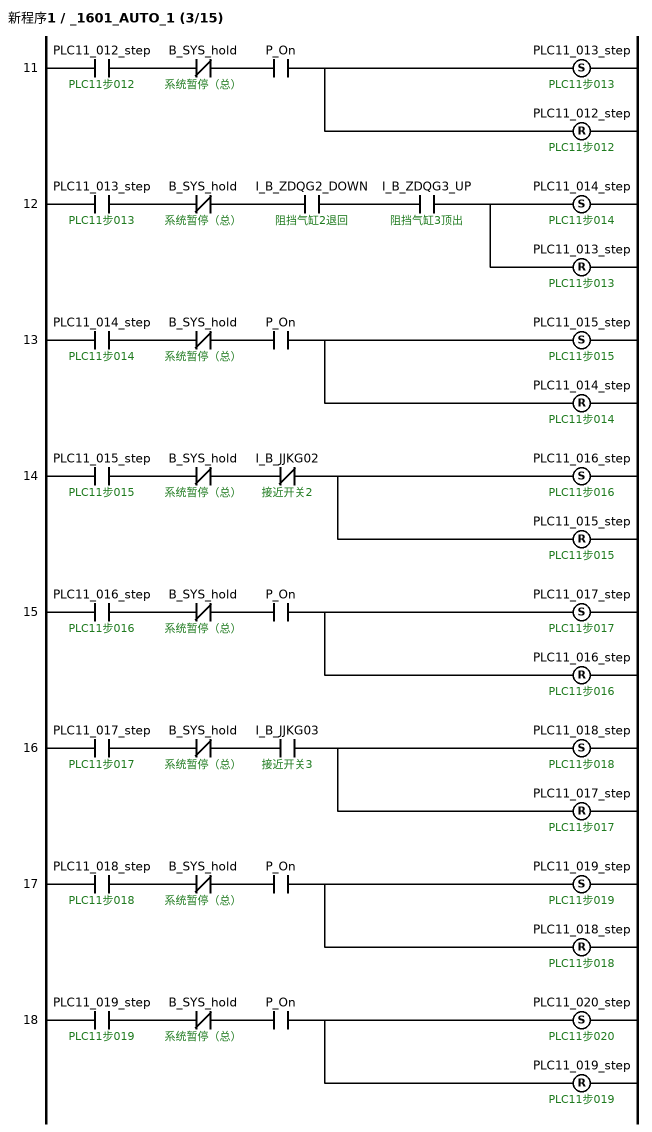
; [picture p24: 新程序1 / _1601_AUTO_1, rungs 11-18]
; rung 11
LD PLC11_012_step  ; PLC11步012
ANDNOT B_SYS_hold  ; 系统暂停（总）
AND P_On
SET PLC11_013_step  ; PLC11步013
RSET PLC11_012_step  ; PLC11步012
; rung 12
LD PLC11_013_step  ; PLC11步013
ANDNOT B_SYS_hold  ; 系统暂停（总）
AND I_B_ZDQG2_DOWN  ; 阻挡气缸2退回
AND I_B_ZDQG3_UP  ; 阻挡气缸3顶出
SET PLC11_014_step  ; PLC11步014
RSET PLC11_013_step  ; PLC11步013
; rung 13
LD PLC11_014_step  ; PLC11步014
ANDNOT B_SYS_hold  ; 系统暂停（总）
AND P_On
SET PLC11_015_step  ; PLC11步015
RSET PLC11_014_step  ; PLC11步014
; rung 14
LD PLC11_015_step  ; PLC11步015
ANDNOT B_SYS_hold  ; 系统暂停（总）
ANDNOT I_B_JJKG02  ; 接近开关2
SET PLC11_016_step  ; PLC11步016
RSET PLC11_015_step  ; PLC11步015
; rung 15
LD PLC11_016_step  ; PLC11步016
ANDNOT B_SYS_hold  ; 系统暂停（总）
AND P_On
SET PLC11_017_step  ; PLC11步017
RSET PLC11_016_step  ; PLC11步016
; rung 16
LD PLC11_017_step  ; PLC11步017
ANDNOT B_SYS_hold  ; 系统暂停（总）
AND I_B_JJKG03  ; 接近开关3
SET PLC11_018_step  ; PLC11步018
RSET PLC11_017_step  ; PLC11步017
; rung 17
LD PLC11_018_step  ; PLC11步018
ANDNOT B_SYS_hold  ; 系统暂停（总）
AND P_On
SET PLC11_019_step  ; PLC11步019
RSET PLC11_018_step  ; PLC11步018
; rung 18
LD PLC11_019_step  ; PLC11步019
ANDNOT B_SYS_hold  ; 系统暂停（总）
AND P_On
SET PLC11_020_step  ; PLC11步020
RSET PLC11_019_step  ; PLC11步019

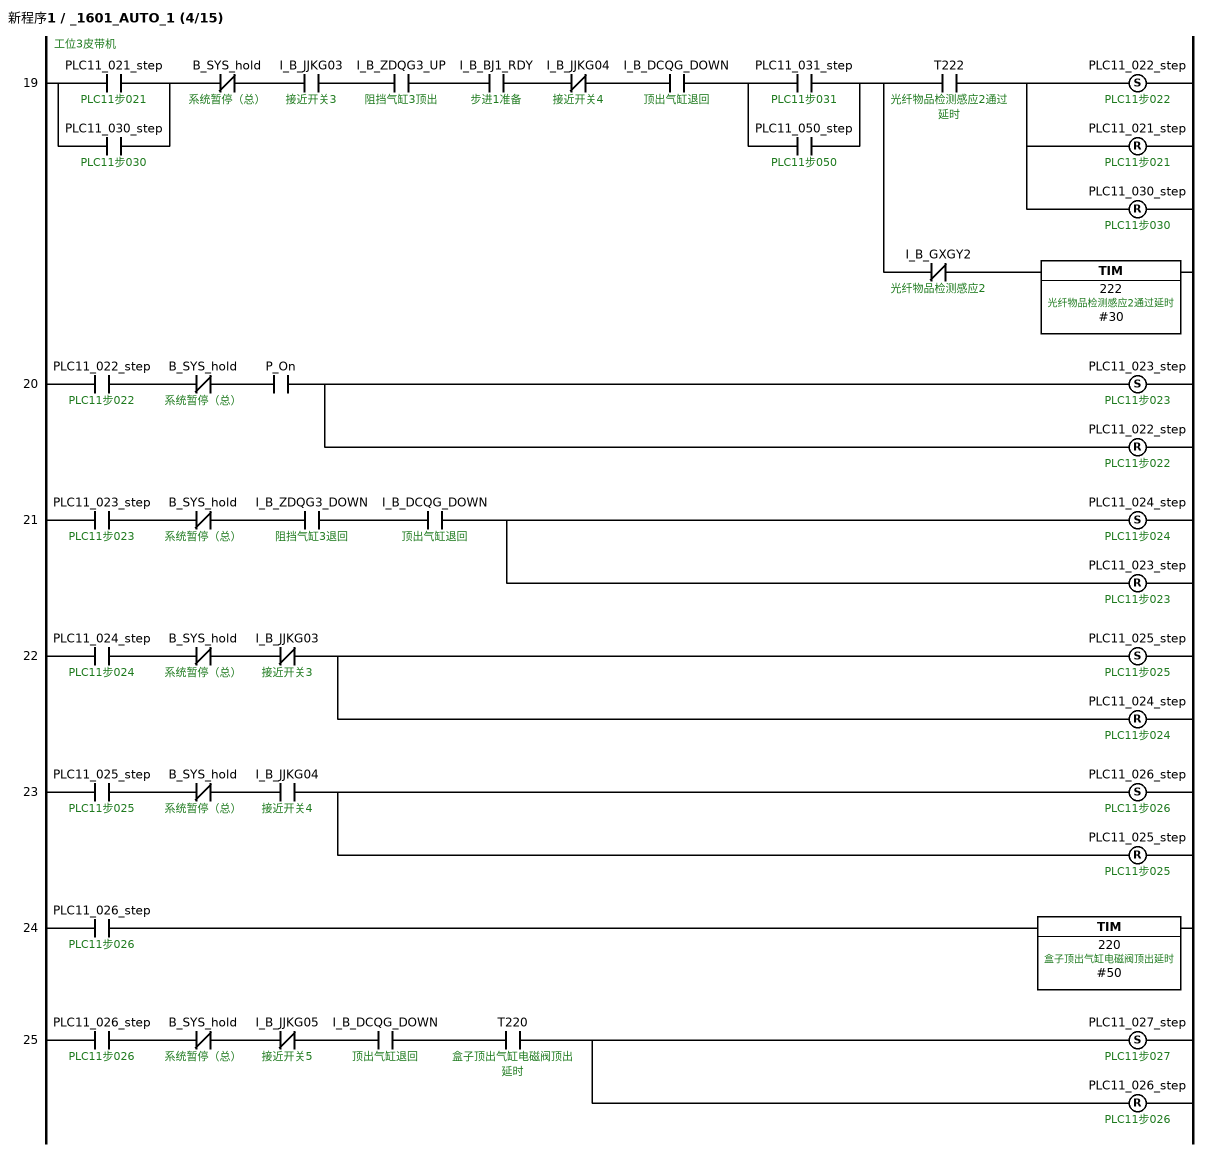
; rung 19: 工位3皮带机
LD PLC11_021_step  ; PLC11步021
OR PLC11_030_step  ; PLC11步030
ANDNOT B_SYS_hold  ; 系统暂停（总）
AND I_B_JJKG03  ; 接近开关3
AND I_B_ZDQG3_UP  ; 阻挡气缸3顶出
AND I_B_BJ1_RDY  ; 步进1准备
ANDNOT I_B_JJKG04  ; 接近开关4
AND I_B_DCQG_DOWN  ; 顶出气缸退回
LD PLC11_031_step  ; PLC11步031
OR PLC11_050_step  ; PLC11步050
ANDLD
OUT TR0
AND T222  ; 光纤物品检测感应2通过延时
SET PLC11_022_step  ; PLC11步022
RSET PLC11_021_step  ; PLC11步021
RSET PLC11_030_step  ; PLC11步030
LD TR0
ANDNOT I_B_GXGY2  ; 光纤物品检测感应2
TIM 222 #30  ; 光纤物品检测感应2通过延时
; rung 20
LD PLC11_022_step  ; PLC11步022
ANDNOT B_SYS_hold  ; 系统暂停（总）
AND P_On
SET PLC11_023_step  ; PLC11步023
RSET PLC11_022_step  ; PLC11步022
; rung 21
LD PLC11_023_step  ; PLC11步023
ANDNOT B_SYS_hold  ; 系统暂停（总）
AND I_B_ZDQG3_DOWN  ; 阻挡气缸3退回
AND I_B_DCQG_DOWN  ; 顶出气缸退回
SET PLC11_024_step  ; PLC11步024
RSET PLC11_023_step  ; PLC11步023
; rung 22
LD PLC11_024_step  ; PLC11步024
ANDNOT B_SYS_hold  ; 系统暂停（总）
ANDNOT I_B_JJKG03  ; 接近开关3
SET PLC11_025_step  ; PLC11步025
RSET PLC11_024_step  ; PLC11步024
; rung 23
LD PLC11_025_step  ; PLC11步025
ANDNOT B_SYS_hold  ; 系统暂停（总）
AND I_B_JJKG04  ; 接近开关4
SET PLC11_026_step  ; PLC11步026
RSET PLC11_025_step  ; PLC11步025
; rung 24
LD PLC11_026_step  ; PLC11步026
TIM 220 #50  ; 盒子顶出气缸电磁阀顶出延时
; rung 25
LD PLC11_026_step  ; PLC11步026
ANDNOT B_SYS_hold  ; 系统暂停（总）
ANDNOT I_B_JJKG05  ; 接近开关5
AND I_B_DCQG_DOWN  ; 顶出气缸退回
AND T220  ; 盒子顶出气缸电磁阀顶出延时
SET PLC11_027_step  ; PLC11步027
RSET PLC11_026_step  ; PLC11步026

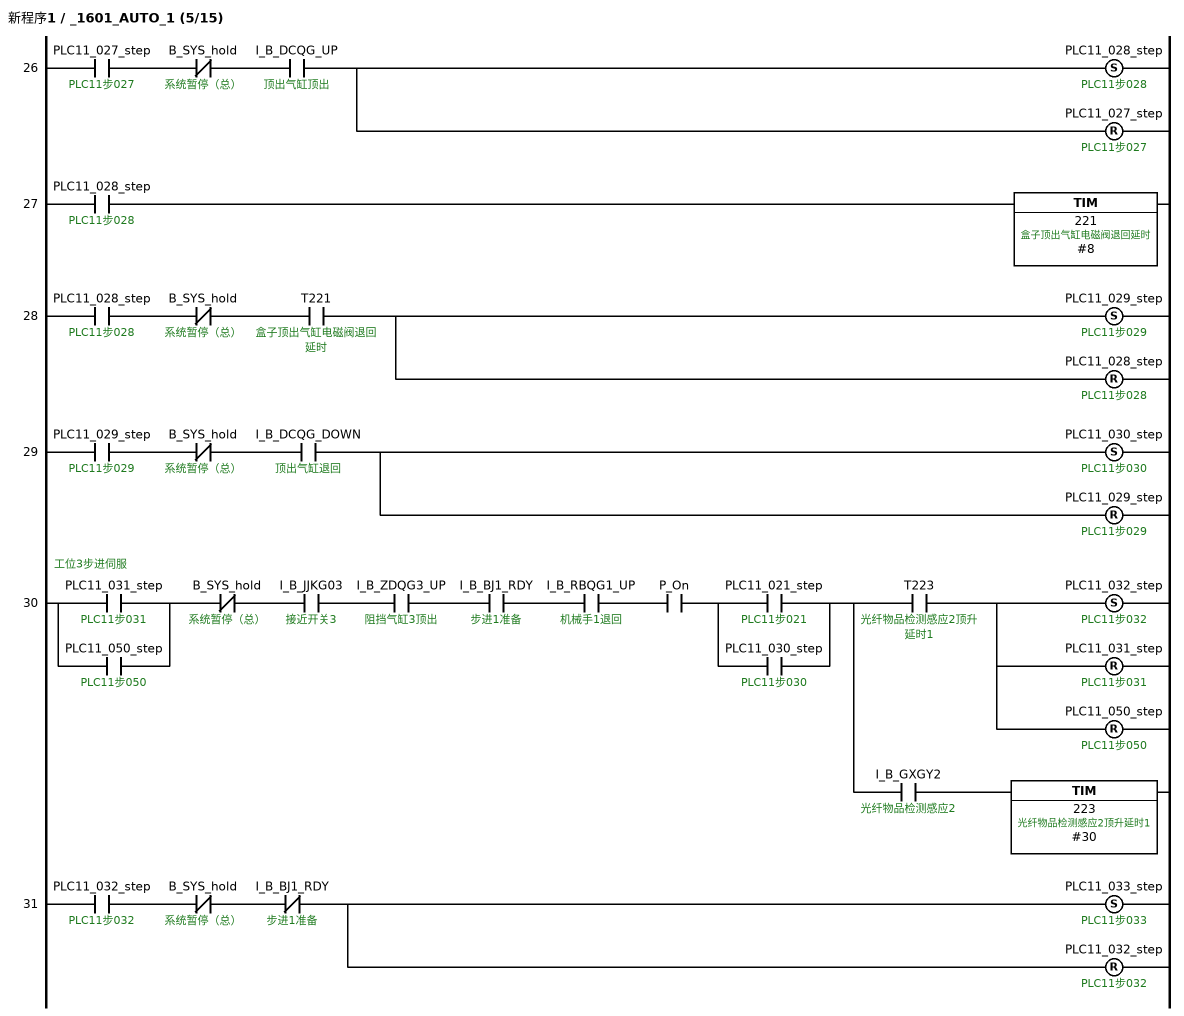
; rung 26
LD PLC11_027_step  ; PLC11步027
ANDNOT B_SYS_hold  ; 系统暂停（总）
AND I_B_DCQG_UP  ; 顶出气缸顶出
SET PLC11_028_step  ; PLC11步028
RSET PLC11_027_step  ; PLC11步027
; rung 27
LD PLC11_028_step  ; PLC11步028
TIM 221 #8  ; 盒子顶出气缸电磁阀退回延时
; rung 28
LD PLC11_028_step  ; PLC11步028
ANDNOT B_SYS_hold  ; 系统暂停（总）
AND T221  ; 盒子顶出气缸电磁阀退回延时
SET PLC11_029_step  ; PLC11步029
RSET PLC11_028_step  ; PLC11步028
; rung 29
LD PLC11_029_step  ; PLC11步029
ANDNOT B_SYS_hold  ; 系统暂停（总）
AND I_B_DCQG_DOWN  ; 顶出气缸退回
SET PLC11_030_step  ; PLC11步030
RSET PLC11_029_step  ; PLC11步029
; rung 30: 工位3步进伺服
LD PLC11_031_step  ; PLC11步031
OR PLC11_050_step  ; PLC11步050
ANDNOT B_SYS_hold  ; 系统暂停（总）
AND I_B_JJKG03  ; 接近开关3
AND I_B_ZDQG3_UP  ; 阻挡气缸3顶出
AND I_B_BJ1_RDY  ; 步进1准备
AND I_B_RBQG1_UP  ; 机械手1退回
AND P_On
LD PLC11_021_step  ; PLC11步021
OR PLC11_030_step  ; PLC11步030
ANDLD
OUT TR0
AND T223  ; 光纤物品检测感应2顶升延时1
SET PLC11_032_step  ; PLC11步032
RSET PLC11_031_step  ; PLC11步031
RSET PLC11_050_step  ; PLC11步050
LD TR0
AND I_B_GXGY2  ; 光纤物品检测感应2
TIM 223 #30  ; 光纤物品检测感应2顶升延时1
; rung 31
LD PLC11_032_step  ; PLC11步032
ANDNOT B_SYS_hold  ; 系统暂停（总）
ANDNOT I_B_BJ1_RDY  ; 步进1准备
SET PLC11_033_step  ; PLC11步033
RSET PLC11_032_step  ; PLC11步032

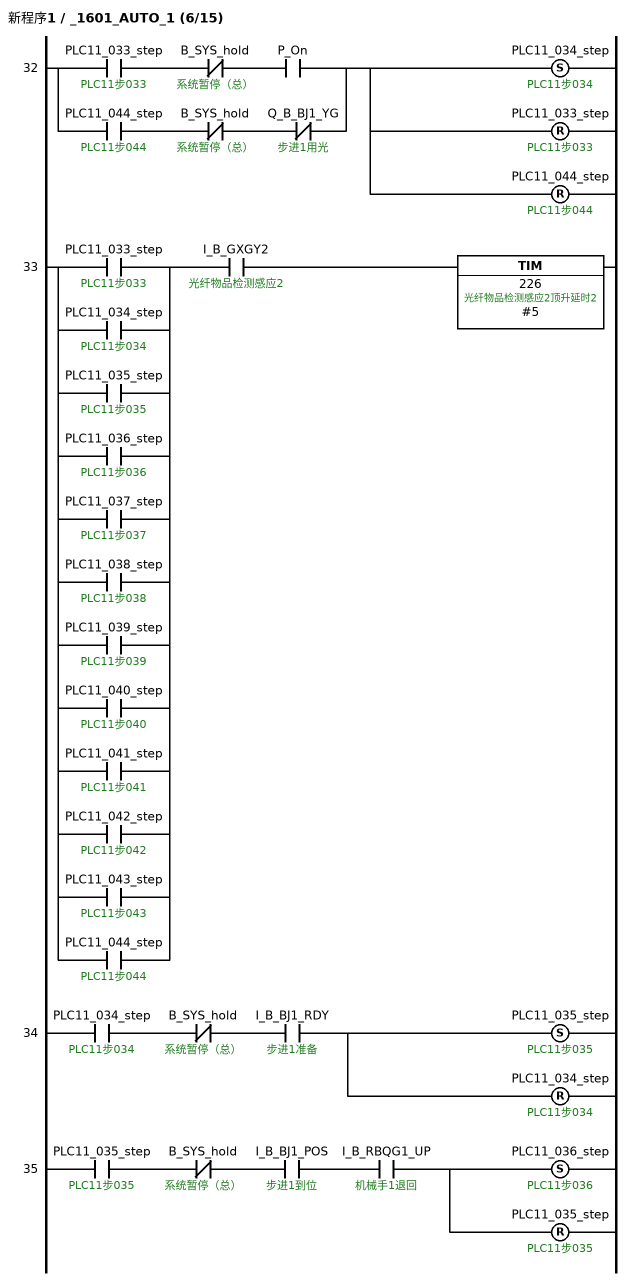
; rung 32
LD PLC11_033_step  ; PLC11步033
ANDNOT B_SYS_hold  ; 系统暂停（总）
AND P_On
LD PLC11_044_step  ; PLC11步044
ANDNOT B_SYS_hold  ; 系统暂停（总）
ANDNOT Q_B_BJ1_YG  ; 步进1用光
ORLD
SET PLC11_034_step  ; PLC11步034
RSET PLC11_033_step  ; PLC11步033
RSET PLC11_044_step  ; PLC11步044
; rung 33
LD PLC11_033_step  ; PLC11步033
OR PLC11_034_step  ; PLC11步034
OR PLC11_035_step  ; PLC11步035
OR PLC11_036_step  ; PLC11步036
OR PLC11_037_step  ; PLC11步037
OR PLC11_038_step  ; PLC11步038
OR PLC11_039_step  ; PLC11步039
OR PLC11_040_step  ; PLC11步040
OR PLC11_041_step  ; PLC11步041
OR PLC11_042_step  ; PLC11步042
OR PLC11_043_step  ; PLC11步043
OR PLC11_044_step  ; PLC11步044
AND I_B_GXGY2  ; 光纤物品检测感应2
TIM 226 #5  ; 光纤物品检测感应2顶升延时2
; rung 34
LD PLC11_034_step  ; PLC11步034
ANDNOT B_SYS_hold  ; 系统暂停（总）
AND I_B_BJ1_RDY  ; 步进1准备
SET PLC11_035_step  ; PLC11步035
RSET PLC11_034_step  ; PLC11步034
; rung 35
LD PLC11_035_step  ; PLC11步035
ANDNOT B_SYS_hold  ; 系统暂停（总）
AND I_B_BJ1_POS  ; 步进1到位
AND I_B_RBQG1_UP  ; 机械手1退回
SET PLC11_036_step  ; PLC11步036
RSET PLC11_035_step  ; PLC11步035

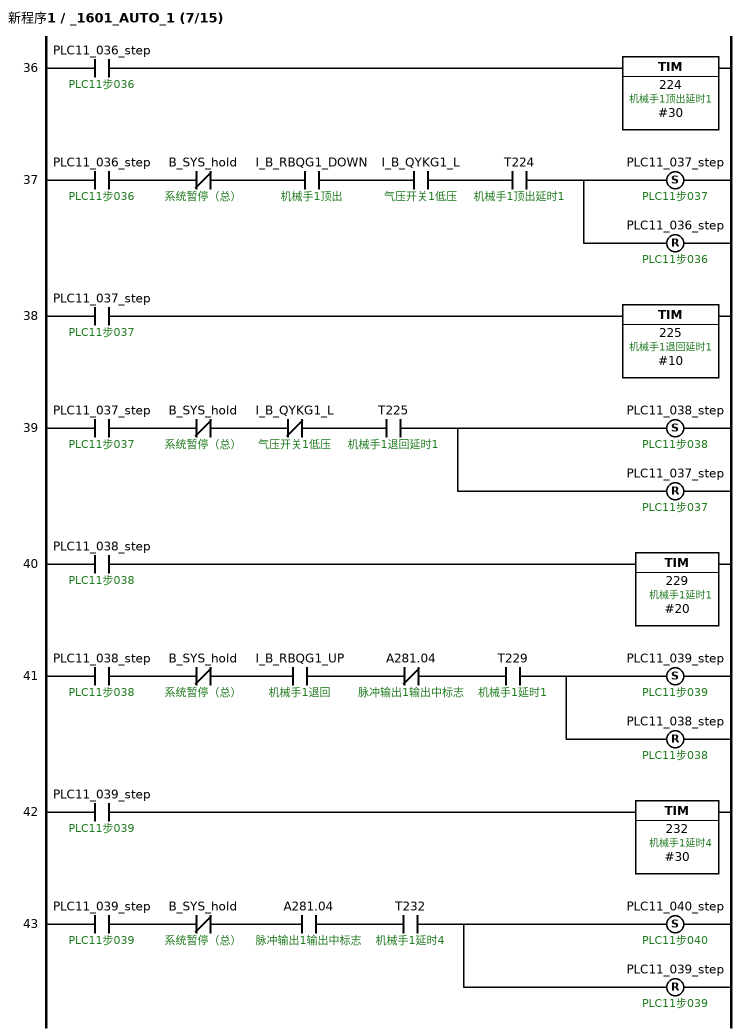
; rung 36
LD PLC11_036_step  ; PLC11步036
TIM 224 #30  ; 机械手1顶出延时1
; rung 37
LD PLC11_036_step  ; PLC11步036
ANDNOT B_SYS_hold  ; 系统暂停（总）
AND I_B_RBQG1_DOWN  ; 机械手1顶出
AND I_B_QYKG1_L  ; 气压开关1低压
AND T224  ; 机械手1顶出延时1
SET PLC11_037_step  ; PLC11步037
RSET PLC11_036_step  ; PLC11步036
; rung 38
LD PLC11_037_step  ; PLC11步037
TIM 225 #10  ; 机械手1退回延时1
; rung 39
LD PLC11_037_step  ; PLC11步037
ANDNOT B_SYS_hold  ; 系统暂停（总）
ANDNOT I_B_QYKG1_L  ; 气压开关1低压
AND T225  ; 机械手1退回延时1
SET PLC11_038_step  ; PLC11步038
RSET PLC11_037_step  ; PLC11步037
; rung 40
LD PLC11_038_step  ; PLC11步038
TIM 229 #20  ; 机械手1延时1
; rung 41
LD PLC11_038_step  ; PLC11步038
ANDNOT B_SYS_hold  ; 系统暂停（总）
AND I_B_RBQG1_UP  ; 机械手1退回
ANDNOT A281.04  ; 脉冲输出1输出中标志
AND T229  ; 机械手1延时1
SET PLC11_039_step  ; PLC11步039
RSET PLC11_038_step  ; PLC11步038
; rung 42
LD PLC11_039_step  ; PLC11步039
TIM 232 #30  ; 机械手1延时4
; rung 43
LD PLC11_039_step  ; PLC11步039
ANDNOT B_SYS_hold  ; 系统暂停（总）
AND A281.04  ; 脉冲输出1输出中标志
AND T232  ; 机械手1延时4
SET PLC11_040_step  ; PLC11步040
RSET PLC11_039_step  ; PLC11步039

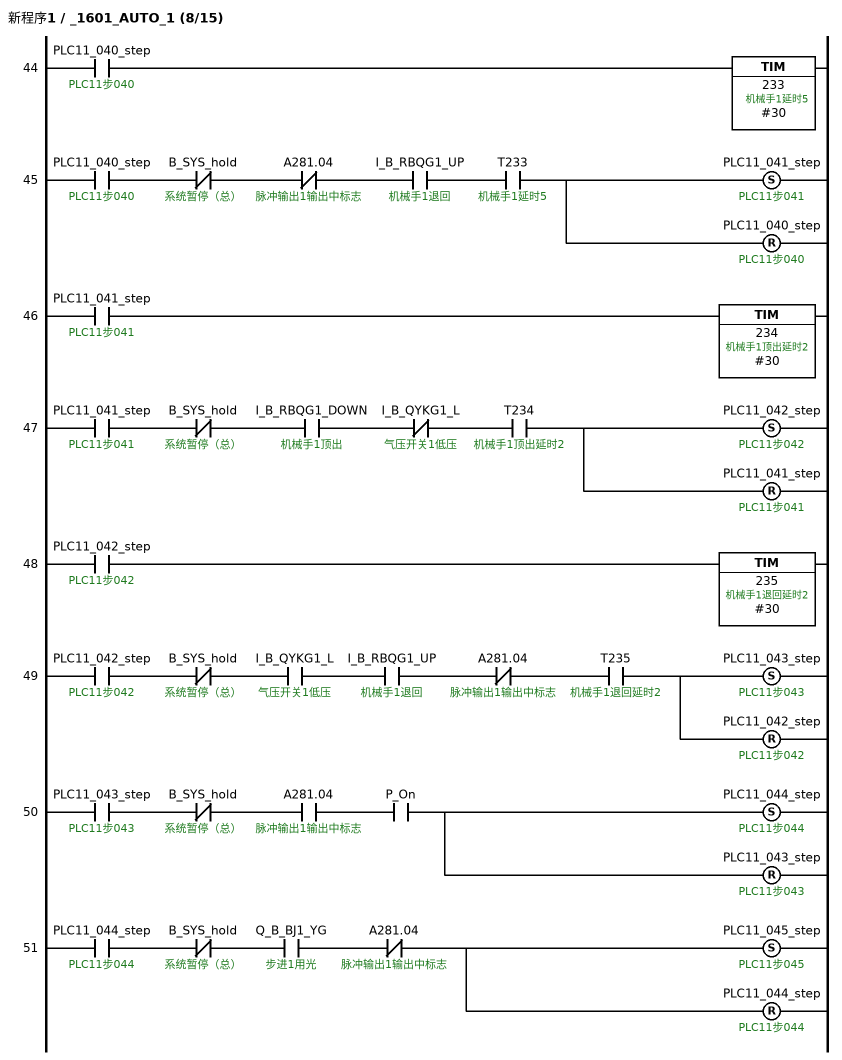
; rung 44
LD PLC11_040_step  ; PLC11步040
TIM 233 #30  ; 机械手1延时5
; rung 45
LD PLC11_040_step  ; PLC11步040
ANDNOT B_SYS_hold  ; 系统暂停（总）
ANDNOT A281.04  ; 脉冲输出1输出中标志
AND I_B_RBQG1_UP  ; 机械手1退回
AND T233  ; 机械手1延时5
SET PLC11_041_step  ; PLC11步041
RSET PLC11_040_step  ; PLC11步040
; rung 46
LD PLC11_041_step  ; PLC11步041
TIM 234 #30  ; 机械手1顶出延时2
; rung 47
LD PLC11_041_step  ; PLC11步041
ANDNOT B_SYS_hold  ; 系统暂停（总）
AND I_B_RBQG1_DOWN  ; 机械手1顶出
ANDNOT I_B_QYKG1_L  ; 气压开关1低压
AND T234  ; 机械手1顶出延时2
SET PLC11_042_step  ; PLC11步042
RSET PLC11_041_step  ; PLC11步041
; rung 48
LD PLC11_042_step  ; PLC11步042
TIM 235 #30  ; 机械手1退回延时2
; rung 49
LD PLC11_042_step  ; PLC11步042
ANDNOT B_SYS_hold  ; 系统暂停（总）
AND I_B_QYKG1_L  ; 气压开关1低压
AND I_B_RBQG1_UP  ; 机械手1退回
ANDNOT A281.04  ; 脉冲输出1输出中标志
AND T235  ; 机械手1退回延时2
SET PLC11_043_step  ; PLC11步043
RSET PLC11_042_step  ; PLC11步042
; rung 50
LD PLC11_043_step  ; PLC11步043
ANDNOT B_SYS_hold  ; 系统暂停（总）
AND A281.04  ; 脉冲输出1输出中标志
AND P_On
SET PLC11_044_step  ; PLC11步044
RSET PLC11_043_step  ; PLC11步043
; rung 51
LD PLC11_044_step  ; PLC11步044
ANDNOT B_SYS_hold  ; 系统暂停（总）
AND Q_B_BJ1_YG  ; 步进1用光
ANDNOT A281.04  ; 脉冲输出1输出中标志
SET PLC11_045_step  ; PLC11步045
RSET PLC11_044_step  ; PLC11步044

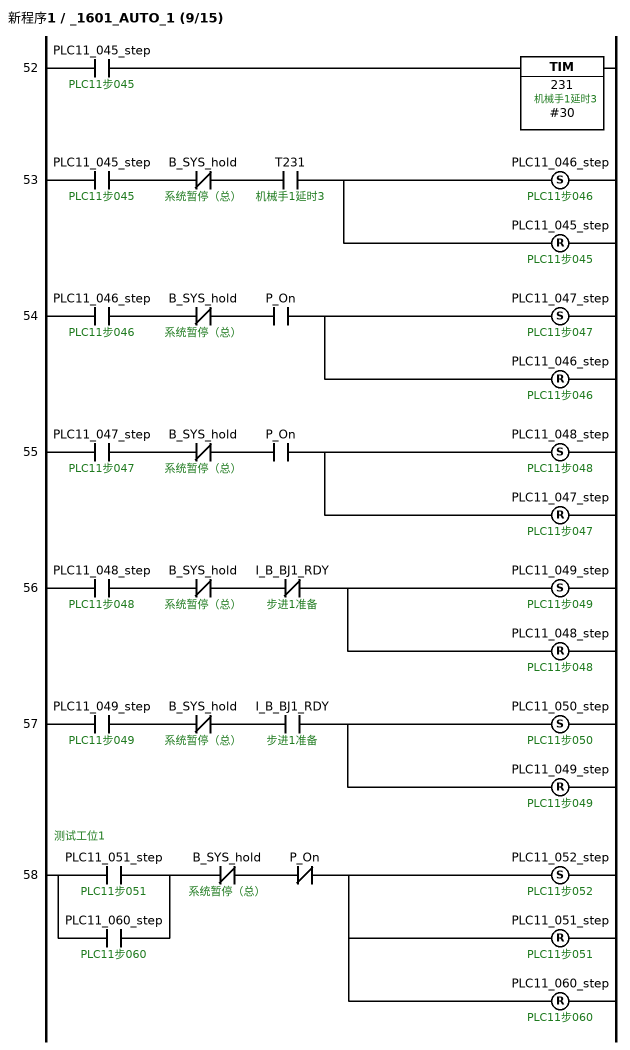
; rung 52
LD PLC11_045_step  ; PLC11步045
TIM 231 #30  ; 机械手1延时3
; rung 53
LD PLC11_045_step  ; PLC11步045
ANDNOT B_SYS_hold  ; 系统暂停（总）
AND T231  ; 机械手1延时3
SET PLC11_046_step  ; PLC11步046
RSET PLC11_045_step  ; PLC11步045
; rung 54
LD PLC11_046_step  ; PLC11步046
ANDNOT B_SYS_hold  ; 系统暂停（总）
AND P_On
SET PLC11_047_step  ; PLC11步047
RSET PLC11_046_step  ; PLC11步046
; rung 55
LD PLC11_047_step  ; PLC11步047
ANDNOT B_SYS_hold  ; 系统暂停（总）
AND P_On
SET PLC11_048_step  ; PLC11步048
RSET PLC11_047_step  ; PLC11步047
; rung 56
LD PLC11_048_step  ; PLC11步048
ANDNOT B_SYS_hold  ; 系统暂停（总）
ANDNOT I_B_BJ1_RDY  ; 步进1准备
SET PLC11_049_step  ; PLC11步049
RSET PLC11_048_step  ; PLC11步048
; rung 57
LD PLC11_049_step  ; PLC11步049
ANDNOT B_SYS_hold  ; 系统暂停（总）
AND I_B_BJ1_RDY  ; 步进1准备
SET PLC11_050_step  ; PLC11步050
RSET PLC11_049_step  ; PLC11步049
; rung 58: 测试工位1
LD PLC11_051_step  ; PLC11步051
OR PLC11_060_step  ; PLC11步060
ANDNOT B_SYS_hold  ; 系统暂停（总）
ANDNOT P_On
SET PLC11_052_step  ; PLC11步052
RSET PLC11_051_step  ; PLC11步051
RSET PLC11_060_step  ; PLC11步060

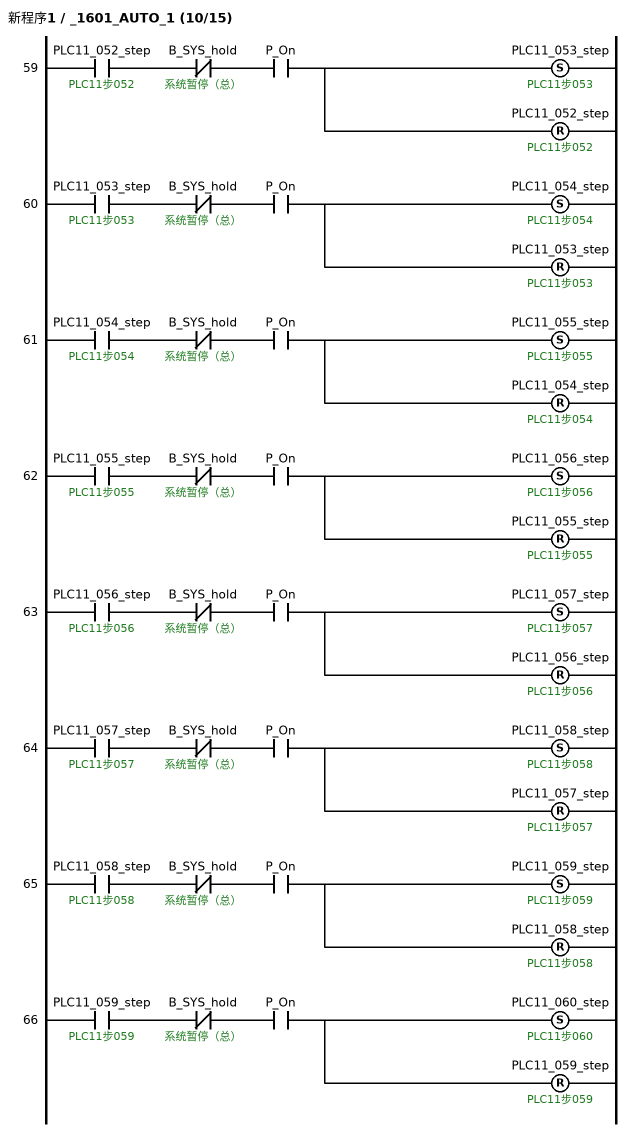
; rung 59
LD PLC11_052_step  ; PLC11步052
ANDNOT B_SYS_hold  ; 系统暂停（总）
AND P_On
SET PLC11_053_step  ; PLC11步053
RSET PLC11_052_step  ; PLC11步052
; rung 60
LD PLC11_053_step  ; PLC11步053
ANDNOT B_SYS_hold  ; 系统暂停（总）
AND P_On
SET PLC11_054_step  ; PLC11步054
RSET PLC11_053_step  ; PLC11步053
; rung 61
LD PLC11_054_step  ; PLC11步054
ANDNOT B_SYS_hold  ; 系统暂停（总）
AND P_On
SET PLC11_055_step  ; PLC11步055
RSET PLC11_054_step  ; PLC11步054
; rung 62
LD PLC11_055_step  ; PLC11步055
ANDNOT B_SYS_hold  ; 系统暂停（总）
AND P_On
SET PLC11_056_step  ; PLC11步056
RSET PLC11_055_step  ; PLC11步055
; rung 63
LD PLC11_056_step  ; PLC11步056
ANDNOT B_SYS_hold  ; 系统暂停（总）
AND P_On
SET PLC11_057_step  ; PLC11步057
RSET PLC11_056_step  ; PLC11步056
; rung 64
LD PLC11_057_step  ; PLC11步057
ANDNOT B_SYS_hold  ; 系统暂停（总）
AND P_On
SET PLC11_058_step  ; PLC11步058
RSET PLC11_057_step  ; PLC11步057
; rung 65
LD PLC11_058_step  ; PLC11步058
ANDNOT B_SYS_hold  ; 系统暂停（总）
AND P_On
SET PLC11_059_step  ; PLC11步059
RSET PLC11_058_step  ; PLC11步058
; rung 66
LD PLC11_059_step  ; PLC11步059
ANDNOT B_SYS_hold  ; 系统暂停（总）
AND P_On
SET PLC11_060_step  ; PLC11步060
RSET PLC11_059_step  ; PLC11步059

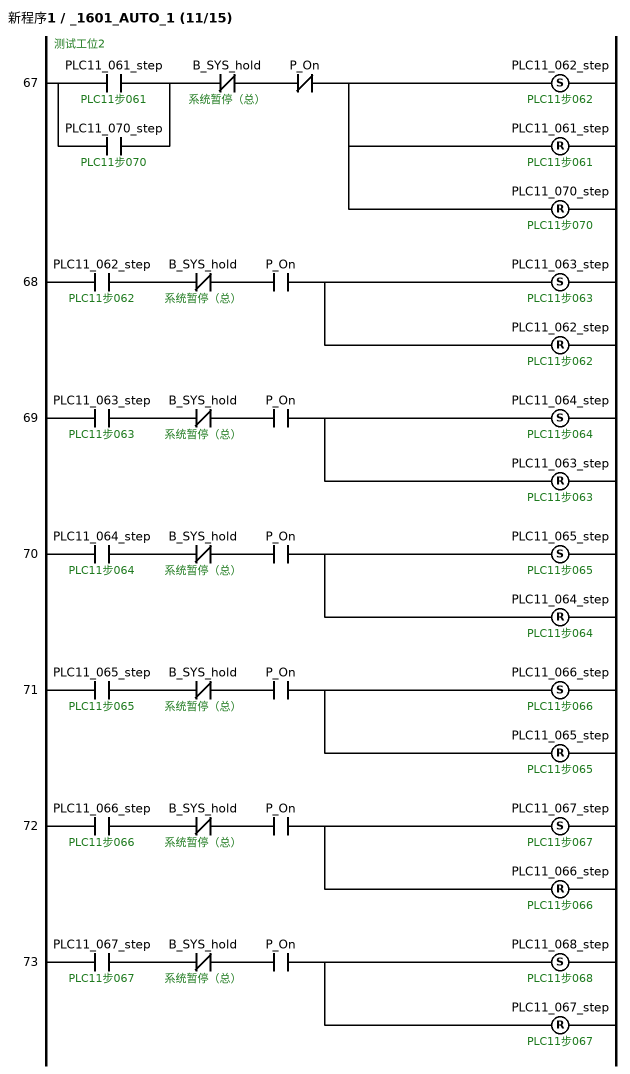
; rung 67: 测试工位2
LD PLC11_061_step  ; PLC11步061
OR PLC11_070_step  ; PLC11步070
ANDNOT B_SYS_hold  ; 系统暂停（总）
ANDNOT P_On
SET PLC11_062_step  ; PLC11步062
RSET PLC11_061_step  ; PLC11步061
RSET PLC11_070_step  ; PLC11步070
; rung 68
LD PLC11_062_step  ; PLC11步062
ANDNOT B_SYS_hold  ; 系统暂停（总）
AND P_On
SET PLC11_063_step  ; PLC11步063
RSET PLC11_062_step  ; PLC11步062
; rung 69
LD PLC11_063_step  ; PLC11步063
ANDNOT B_SYS_hold  ; 系统暂停（总）
AND P_On
SET PLC11_064_step  ; PLC11步064
RSET PLC11_063_step  ; PLC11步063
; rung 70
LD PLC11_064_step  ; PLC11步064
ANDNOT B_SYS_hold  ; 系统暂停（总）
AND P_On
SET PLC11_065_step  ; PLC11步065
RSET PLC11_064_step  ; PLC11步064
; rung 71
LD PLC11_065_step  ; PLC11步065
ANDNOT B_SYS_hold  ; 系统暂停（总）
AND P_On
SET PLC11_066_step  ; PLC11步066
RSET PLC11_065_step  ; PLC11步065
; rung 72
LD PLC11_066_step  ; PLC11步066
ANDNOT B_SYS_hold  ; 系统暂停（总）
AND P_On
SET PLC11_067_step  ; PLC11步067
RSET PLC11_066_step  ; PLC11步066
; rung 73
LD PLC11_067_step  ; PLC11步067
ANDNOT B_SYS_hold  ; 系统暂停（总）
AND P_On
SET PLC11_068_step  ; PLC11步068
RSET PLC11_067_step  ; PLC11步067

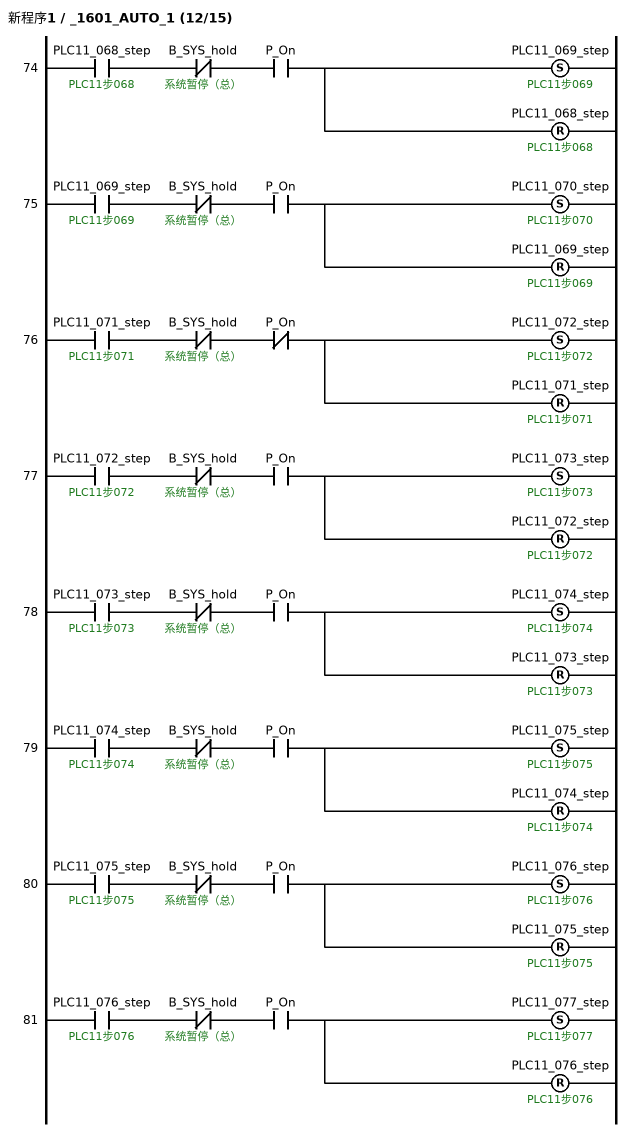
; rung 74
LD PLC11_068_step  ; PLC11步068
ANDNOT B_SYS_hold  ; 系统暂停（总）
AND P_On
SET PLC11_069_step  ; PLC11步069
RSET PLC11_068_step  ; PLC11步068
; rung 75
LD PLC11_069_step  ; PLC11步069
ANDNOT B_SYS_hold  ; 系统暂停（总）
AND P_On
SET PLC11_070_step  ; PLC11步070
RSET PLC11_069_step  ; PLC11步069
; rung 76
LD PLC11_071_step  ; PLC11步071
ANDNOT B_SYS_hold  ; 系统暂停（总）
ANDNOT P_On
SET PLC11_072_step  ; PLC11步072
RSET PLC11_071_step  ; PLC11步071
; rung 77
LD PLC11_072_step  ; PLC11步072
ANDNOT B_SYS_hold  ; 系统暂停（总）
AND P_On
SET PLC11_073_step  ; PLC11步073
RSET PLC11_072_step  ; PLC11步072
; rung 78
LD PLC11_073_step  ; PLC11步073
ANDNOT B_SYS_hold  ; 系统暂停（总）
AND P_On
SET PLC11_074_step  ; PLC11步074
RSET PLC11_073_step  ; PLC11步073
; rung 79
LD PLC11_074_step  ; PLC11步074
ANDNOT B_SYS_hold  ; 系统暂停（总）
AND P_On
SET PLC11_075_step  ; PLC11步075
RSET PLC11_074_step  ; PLC11步074
; rung 80
LD PLC11_075_step  ; PLC11步075
ANDNOT B_SYS_hold  ; 系统暂停（总）
AND P_On
SET PLC11_076_step  ; PLC11步076
RSET PLC11_075_step  ; PLC11步075
; rung 81
LD PLC11_076_step  ; PLC11步076
ANDNOT B_SYS_hold  ; 系统暂停（总）
AND P_On
SET PLC11_077_step  ; PLC11步077
RSET PLC11_076_step  ; PLC11步076

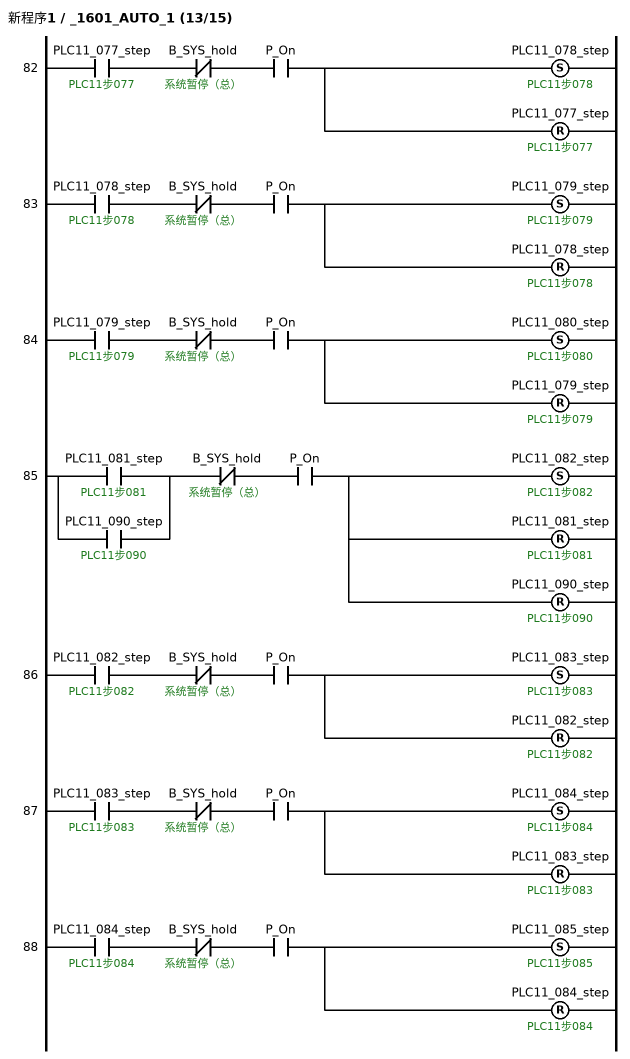
; rung 82
LD PLC11_077_step  ; PLC11步077
ANDNOT B_SYS_hold  ; 系统暂停（总）
AND P_On
SET PLC11_078_step  ; PLC11步078
RSET PLC11_077_step  ; PLC11步077
; rung 83
LD PLC11_078_step  ; PLC11步078
ANDNOT B_SYS_hold  ; 系统暂停（总）
AND P_On
SET PLC11_079_step  ; PLC11步079
RSET PLC11_078_step  ; PLC11步078
; rung 84
LD PLC11_079_step  ; PLC11步079
ANDNOT B_SYS_hold  ; 系统暂停（总）
AND P_On
SET PLC11_080_step  ; PLC11步080
RSET PLC11_079_step  ; PLC11步079
; rung 85
LD PLC11_081_step  ; PLC11步081
OR PLC11_090_step  ; PLC11步090
ANDNOT B_SYS_hold  ; 系统暂停（总）
AND P_On
SET PLC11_082_step  ; PLC11步082
RSET PLC11_081_step  ; PLC11步081
RSET PLC11_090_step  ; PLC11步090
; rung 86
LD PLC11_082_step  ; PLC11步082
ANDNOT B_SYS_hold  ; 系统暂停（总）
AND P_On
SET PLC11_083_step  ; PLC11步083
RSET PLC11_082_step  ; PLC11步082
; rung 87
LD PLC11_083_step  ; PLC11步083
ANDNOT B_SYS_hold  ; 系统暂停（总）
AND P_On
SET PLC11_084_step  ; PLC11步084
RSET PLC11_083_step  ; PLC11步083
; rung 88
LD PLC11_084_step  ; PLC11步084
ANDNOT B_SYS_hold  ; 系统暂停（总）
AND P_On
SET PLC11_085_step  ; PLC11步085
RSET PLC11_084_step  ; PLC11步084

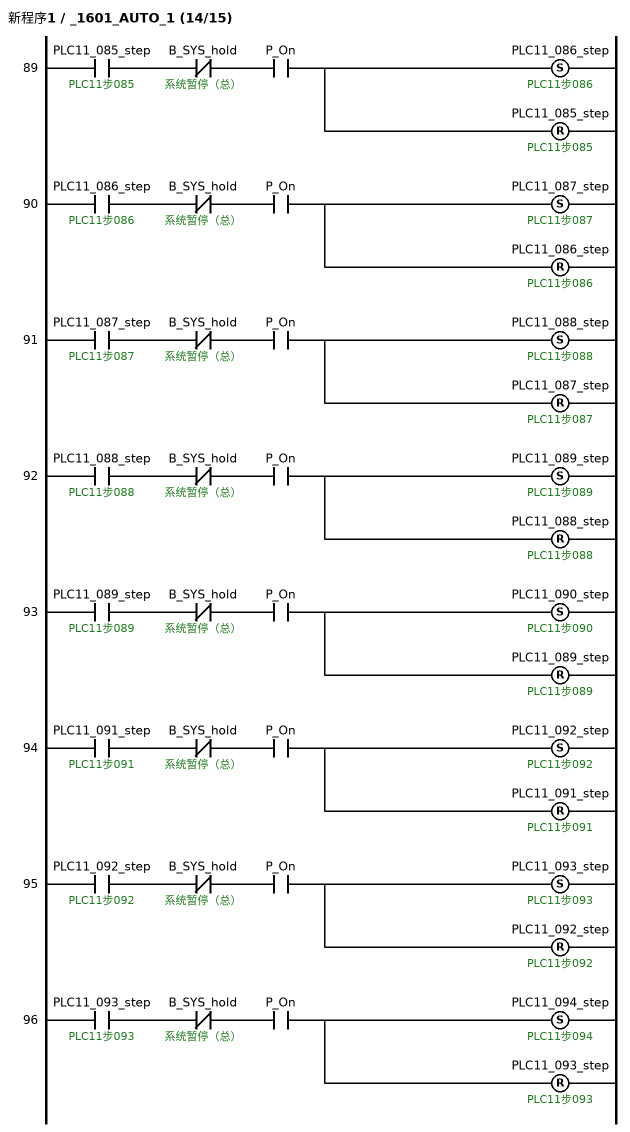
; rung 89
LD PLC11_085_step  ; PLC11步085
ANDNOT B_SYS_hold  ; 系统暂停（总）
AND P_On
SET PLC11_086_step  ; PLC11步086
RSET PLC11_085_step  ; PLC11步085
; rung 90
LD PLC11_086_step  ; PLC11步086
ANDNOT B_SYS_hold  ; 系统暂停（总）
AND P_On
SET PLC11_087_step  ; PLC11步087
RSET PLC11_086_step  ; PLC11步086
; rung 91
LD PLC11_087_step  ; PLC11步087
ANDNOT B_SYS_hold  ; 系统暂停（总）
AND P_On
SET PLC11_088_step  ; PLC11步088
RSET PLC11_087_step  ; PLC11步087
; rung 92
LD PLC11_088_step  ; PLC11步088
ANDNOT B_SYS_hold  ; 系统暂停（总）
AND P_On
SET PLC11_089_step  ; PLC11步089
RSET PLC11_088_step  ; PLC11步088
; rung 93
LD PLC11_089_step  ; PLC11步089
ANDNOT B_SYS_hold  ; 系统暂停（总）
AND P_On
SET PLC11_090_step  ; PLC11步090
RSET PLC11_089_step  ; PLC11步089
; rung 94
LD PLC11_091_step  ; PLC11步091
ANDNOT B_SYS_hold  ; 系统暂停（总）
AND P_On
SET PLC11_092_step  ; PLC11步092
RSET PLC11_091_step  ; PLC11步091
; rung 95
LD PLC11_092_step  ; PLC11步092
ANDNOT B_SYS_hold  ; 系统暂停（总）
AND P_On
SET PLC11_093_step  ; PLC11步093
RSET PLC11_092_step  ; PLC11步092
; rung 96
LD PLC11_093_step  ; PLC11步093
ANDNOT B_SYS_hold  ; 系统暂停（总）
AND P_On
SET PLC11_094_step  ; PLC11步094
RSET PLC11_093_step  ; PLC11步093

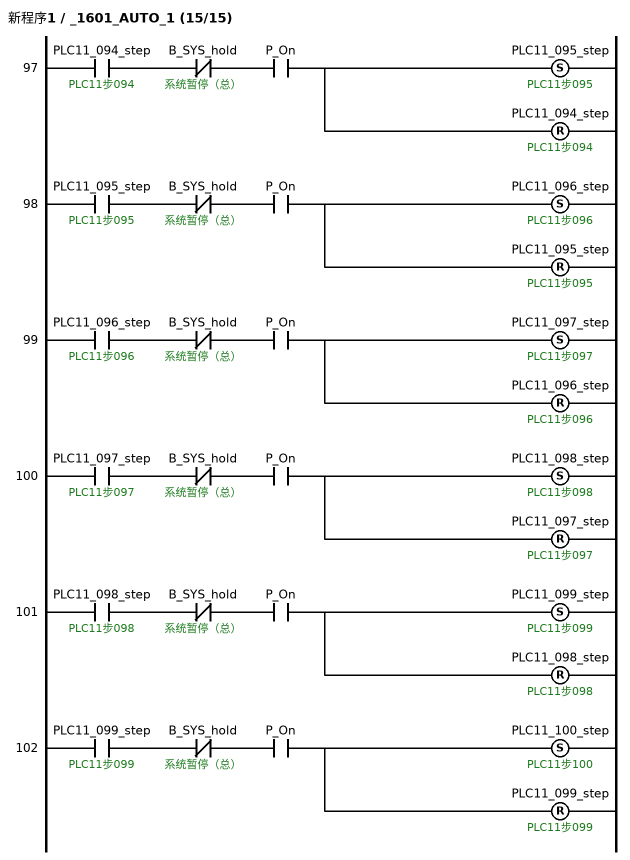
; rung 97
LD PLC11_094_step  ; PLC11步094
ANDNOT B_SYS_hold  ; 系统暂停（总）
AND P_On
SET PLC11_095_step  ; PLC11步095
RSET PLC11_094_step  ; PLC11步094
; rung 98
LD PLC11_095_step  ; PLC11步095
ANDNOT B_SYS_hold  ; 系统暂停（总）
AND P_On
SET PLC11_096_step  ; PLC11步096
RSET PLC11_095_step  ; PLC11步095
; rung 99
LD PLC11_096_step  ; PLC11步096
ANDNOT B_SYS_hold  ; 系统暂停（总）
AND P_On
SET PLC11_097_step  ; PLC11步097
RSET PLC11_096_step  ; PLC11步096
; rung 100
LD PLC11_097_step  ; PLC11步097
ANDNOT B_SYS_hold  ; 系统暂停（总）
AND P_On
SET PLC11_098_step  ; PLC11步098
RSET PLC11_097_step  ; PLC11步097
; rung 101
LD PLC11_098_step  ; PLC11步098
ANDNOT B_SYS_hold  ; 系统暂停（总）
AND P_On
SET PLC11_099_step  ; PLC11步099
RSET PLC11_098_step  ; PLC11步098
; rung 102
LD PLC11_099_step  ; PLC11步099
ANDNOT B_SYS_hold  ; 系统暂停（总）
AND P_On
SET PLC11_100_step  ; PLC11步100
RSET PLC11_099_step  ; PLC11步099

### Section _1601_AUTO_2

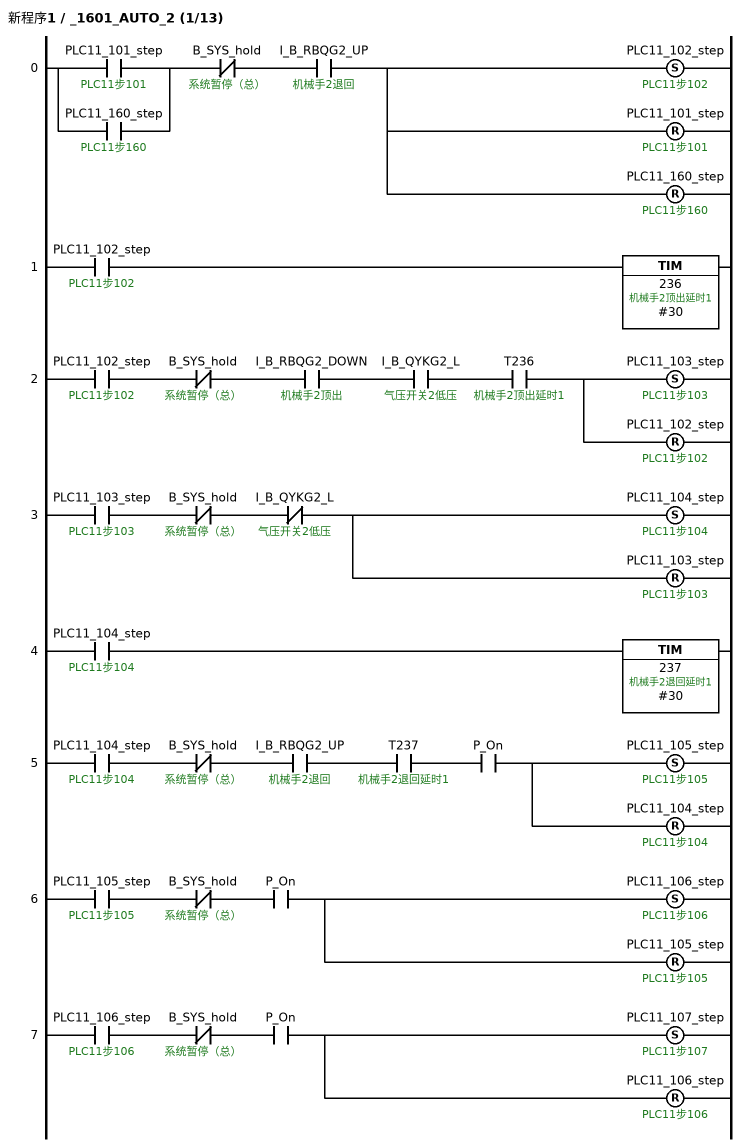
; rung 0
LD PLC11_101_step  ; PLC11步101
OR PLC11_160_step  ; PLC11步160
ANDNOT B_SYS_hold  ; 系统暂停（总）
AND I_B_RBQG2_UP  ; 机械手2退回
SET PLC11_102_step  ; PLC11步102
RSET PLC11_101_step  ; PLC11步101
RSET PLC11_160_step  ; PLC11步160
; rung 1
LD PLC11_102_step  ; PLC11步102
TIM 236 #30  ; 机械手2顶出延时1
; rung 2
LD PLC11_102_step  ; PLC11步102
ANDNOT B_SYS_hold  ; 系统暂停（总）
AND I_B_RBQG2_DOWN  ; 机械手2顶出
AND I_B_QYKG2_L  ; 气压开关2低压
AND T236  ; 机械手2顶出延时1
SET PLC11_103_step  ; PLC11步103
RSET PLC11_102_step  ; PLC11步102
; rung 3
LD PLC11_103_step  ; PLC11步103
ANDNOT B_SYS_hold  ; 系统暂停（总）
ANDNOT I_B_QYKG2_L  ; 气压开关2低压
SET PLC11_104_step  ; PLC11步104
RSET PLC11_103_step  ; PLC11步103
; rung 4
LD PLC11_104_step  ; PLC11步104
TIM 237 #30  ; 机械手2退回延时1
; rung 5
LD PLC11_104_step  ; PLC11步104
ANDNOT B_SYS_hold  ; 系统暂停（总）
AND I_B_RBQG2_UP  ; 机械手2退回
AND T237  ; 机械手2退回延时1
AND P_On
SET PLC11_105_step  ; PLC11步105
RSET PLC11_104_step  ; PLC11步104
; rung 6
LD PLC11_105_step  ; PLC11步105
ANDNOT B_SYS_hold  ; 系统暂停（总）
AND P_On
SET PLC11_106_step  ; PLC11步106
RSET PLC11_105_step  ; PLC11步105
; rung 7
LD PLC11_106_step  ; PLC11步106
ANDNOT B_SYS_hold  ; 系统暂停（总）
AND P_On
SET PLC11_107_step  ; PLC11步107
RSET PLC11_106_step  ; PLC11步106

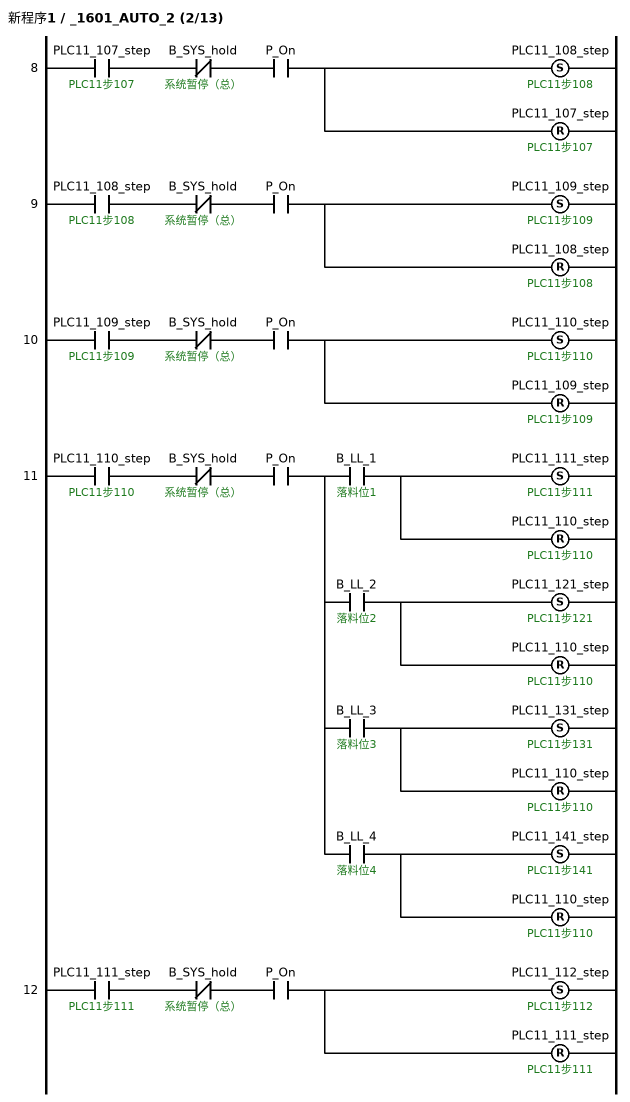
; rung 8
LD PLC11_107_step  ; PLC11步107
ANDNOT B_SYS_hold  ; 系统暂停（总）
AND P_On
SET PLC11_108_step  ; PLC11步108
RSET PLC11_107_step  ; PLC11步107
; rung 9
LD PLC11_108_step  ; PLC11步108
ANDNOT B_SYS_hold  ; 系统暂停（总）
AND P_On
SET PLC11_109_step  ; PLC11步109
RSET PLC11_108_step  ; PLC11步108
; rung 10
LD PLC11_109_step  ; PLC11步109
ANDNOT B_SYS_hold  ; 系统暂停（总）
AND P_On
SET PLC11_110_step  ; PLC11步110
RSET PLC11_109_step  ; PLC11步109
; rung 11
LD PLC11_110_step  ; PLC11步110
ANDNOT B_SYS_hold  ; 系统暂停（总）
AND P_On
OUT TR0
AND B_LL_1  ; 落料位1
SET PLC11_111_step  ; PLC11步111
RSET PLC11_110_step  ; PLC11步110
LD TR0
AND B_LL_2  ; 落料位2
SET PLC11_121_step  ; PLC11步121
RSET PLC11_110_step  ; PLC11步110
LD TR0
AND B_LL_3  ; 落料位3
SET PLC11_131_step  ; PLC11步131
RSET PLC11_110_step  ; PLC11步110
LD TR0
AND B_LL_4  ; 落料位4
SET PLC11_141_step  ; PLC11步141
RSET PLC11_110_step  ; PLC11步110
; rung 12
LD PLC11_111_step  ; PLC11步111
ANDNOT B_SYS_hold  ; 系统暂停（总）
AND P_On
SET PLC11_112_step  ; PLC11步112
RSET PLC11_111_step  ; PLC11步111

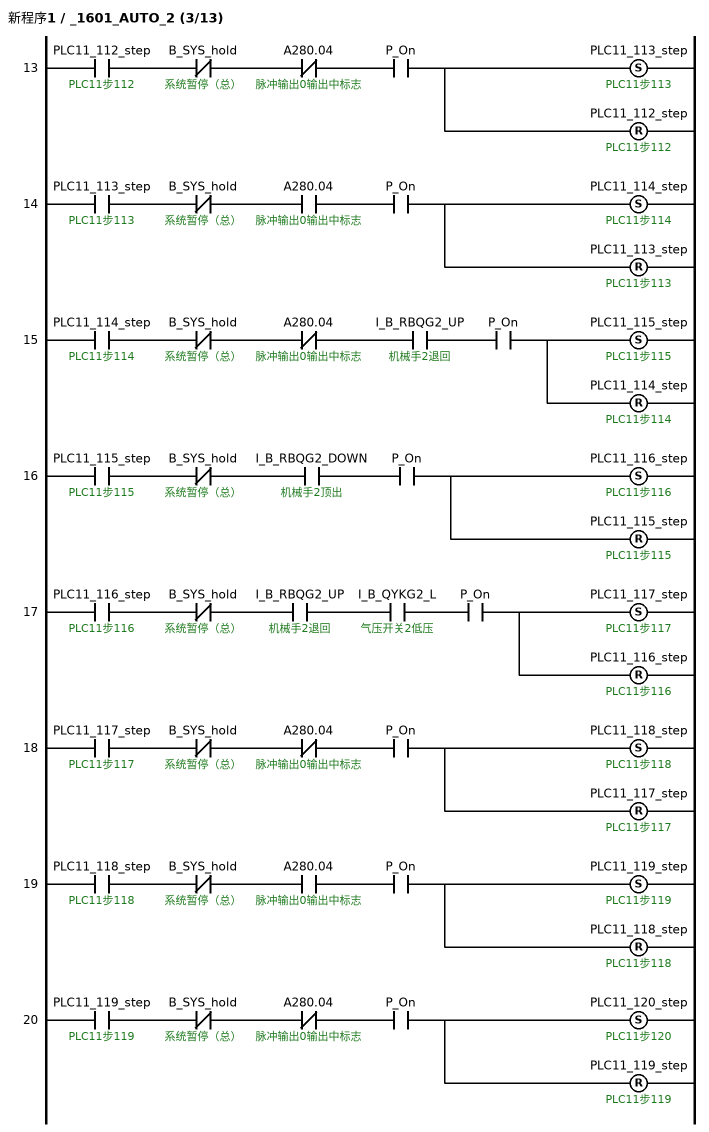
; rung 13
LD PLC11_112_step  ; PLC11步112
ANDNOT B_SYS_hold  ; 系统暂停（总）
ANDNOT A280.04  ; 脉冲输出0输出中标志
AND P_On
SET PLC11_113_step  ; PLC11步113
RSET PLC11_112_step  ; PLC11步112
; rung 14
LD PLC11_113_step  ; PLC11步113
ANDNOT B_SYS_hold  ; 系统暂停（总）
AND A280.04  ; 脉冲输出0输出中标志
AND P_On
SET PLC11_114_step  ; PLC11步114
RSET PLC11_113_step  ; PLC11步113
; rung 15
LD PLC11_114_step  ; PLC11步114
ANDNOT B_SYS_hold  ; 系统暂停（总）
ANDNOT A280.04  ; 脉冲输出0输出中标志
AND I_B_RBQG2_UP  ; 机械手2退回
AND P_On
SET PLC11_115_step  ; PLC11步115
RSET PLC11_114_step  ; PLC11步114
; rung 16
LD PLC11_115_step  ; PLC11步115
ANDNOT B_SYS_hold  ; 系统暂停（总）
AND I_B_RBQG2_DOWN  ; 机械手2顶出
AND P_On
SET PLC11_116_step  ; PLC11步116
RSET PLC11_115_step  ; PLC11步115
; rung 17
LD PLC11_116_step  ; PLC11步116
ANDNOT B_SYS_hold  ; 系统暂停（总）
AND I_B_RBQG2_UP  ; 机械手2退回
AND I_B_QYKG2_L  ; 气压开关2低压
AND P_On
SET PLC11_117_step  ; PLC11步117
RSET PLC11_116_step  ; PLC11步116
; rung 18
LD PLC11_117_step  ; PLC11步117
ANDNOT B_SYS_hold  ; 系统暂停（总）
ANDNOT A280.04  ; 脉冲输出0输出中标志
AND P_On
SET PLC11_118_step  ; PLC11步118
RSET PLC11_117_step  ; PLC11步117
; rung 19
LD PLC11_118_step  ; PLC11步118
ANDNOT B_SYS_hold  ; 系统暂停（总）
AND A280.04  ; 脉冲输出0输出中标志
AND P_On
SET PLC11_119_step  ; PLC11步119
RSET PLC11_118_step  ; PLC11步118
; rung 20
LD PLC11_119_step  ; PLC11步119
ANDNOT B_SYS_hold  ; 系统暂停（总）
ANDNOT A280.04  ; 脉冲输出0输出中标志
AND P_On
SET PLC11_120_step  ; PLC11步120
RSET PLC11_119_step  ; PLC11步119

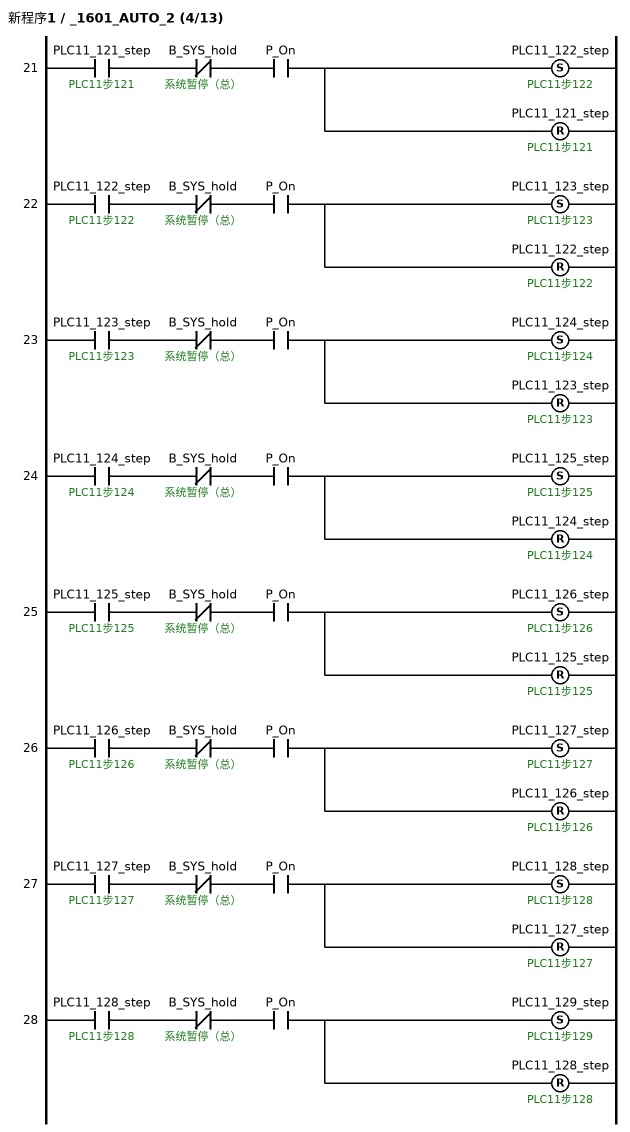
; rung 21
LD PLC11_121_step  ; PLC11步121
ANDNOT B_SYS_hold  ; 系统暂停（总）
AND P_On
SET PLC11_122_step  ; PLC11步122
RSET PLC11_121_step  ; PLC11步121
; rung 22
LD PLC11_122_step  ; PLC11步122
ANDNOT B_SYS_hold  ; 系统暂停（总）
AND P_On
SET PLC11_123_step  ; PLC11步123
RSET PLC11_122_step  ; PLC11步122
; rung 23
LD PLC11_123_step  ; PLC11步123
ANDNOT B_SYS_hold  ; 系统暂停（总）
AND P_On
SET PLC11_124_step  ; PLC11步124
RSET PLC11_123_step  ; PLC11步123
; rung 24
LD PLC11_124_step  ; PLC11步124
ANDNOT B_SYS_hold  ; 系统暂停（总）
AND P_On
SET PLC11_125_step  ; PLC11步125
RSET PLC11_124_step  ; PLC11步124
; rung 25
LD PLC11_125_step  ; PLC11步125
ANDNOT B_SYS_hold  ; 系统暂停（总）
AND P_On
SET PLC11_126_step  ; PLC11步126
RSET PLC11_125_step  ; PLC11步125
; rung 26
LD PLC11_126_step  ; PLC11步126
ANDNOT B_SYS_hold  ; 系统暂停（总）
AND P_On
SET PLC11_127_step  ; PLC11步127
RSET PLC11_126_step  ; PLC11步126
; rung 27
LD PLC11_127_step  ; PLC11步127
ANDNOT B_SYS_hold  ; 系统暂停（总）
AND P_On
SET PLC11_128_step  ; PLC11步128
RSET PLC11_127_step  ; PLC11步127
; rung 28
LD PLC11_128_step  ; PLC11步128
ANDNOT B_SYS_hold  ; 系统暂停（总）
AND P_On
SET PLC11_129_step  ; PLC11步129
RSET PLC11_128_step  ; PLC11步128

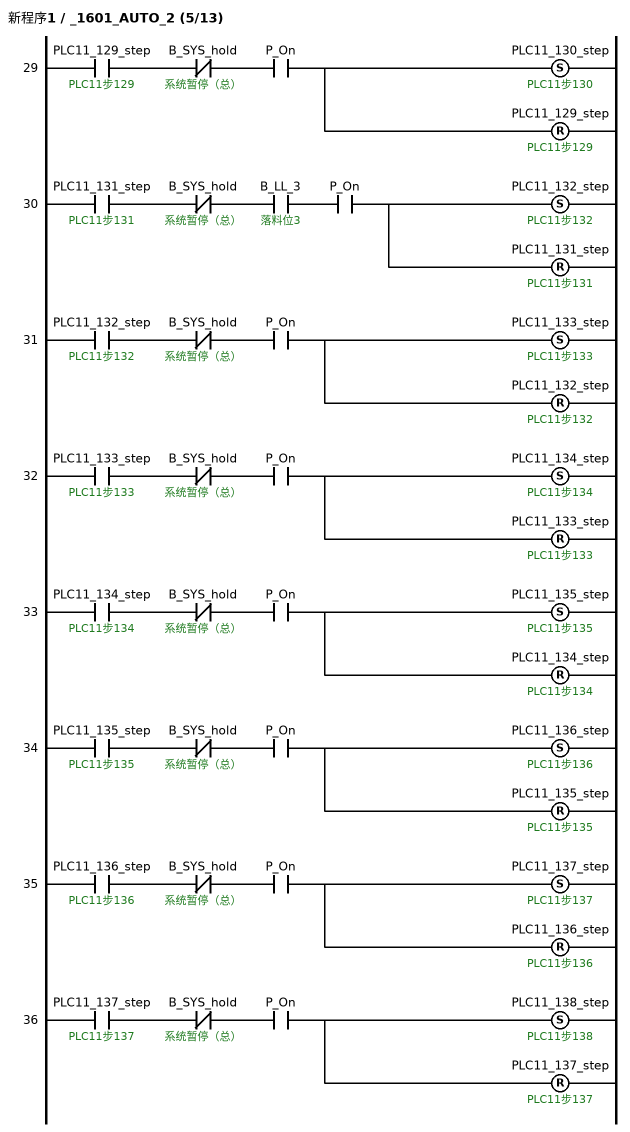
; rung 29
LD PLC11_129_step  ; PLC11步129
ANDNOT B_SYS_hold  ; 系统暂停（总）
AND P_On
SET PLC11_130_step  ; PLC11步130
RSET PLC11_129_step  ; PLC11步129
; rung 30
LD PLC11_131_step  ; PLC11步131
ANDNOT B_SYS_hold  ; 系统暂停（总）
AND B_LL_3  ; 落料位3
AND P_On
SET PLC11_132_step  ; PLC11步132
RSET PLC11_131_step  ; PLC11步131
; rung 31
LD PLC11_132_step  ; PLC11步132
ANDNOT B_SYS_hold  ; 系统暂停（总）
AND P_On
SET PLC11_133_step  ; PLC11步133
RSET PLC11_132_step  ; PLC11步132
; rung 32
LD PLC11_133_step  ; PLC11步133
ANDNOT B_SYS_hold  ; 系统暂停（总）
AND P_On
SET PLC11_134_step  ; PLC11步134
RSET PLC11_133_step  ; PLC11步133
; rung 33
LD PLC11_134_step  ; PLC11步134
ANDNOT B_SYS_hold  ; 系统暂停（总）
AND P_On
SET PLC11_135_step  ; PLC11步135
RSET PLC11_134_step  ; PLC11步134
; rung 34
LD PLC11_135_step  ; PLC11步135
ANDNOT B_SYS_hold  ; 系统暂停（总）
AND P_On
SET PLC11_136_step  ; PLC11步136
RSET PLC11_135_step  ; PLC11步135
; rung 35
LD PLC11_136_step  ; PLC11步136
ANDNOT B_SYS_hold  ; 系统暂停（总）
AND P_On
SET PLC11_137_step  ; PLC11步137
RSET PLC11_136_step  ; PLC11步136
; rung 36
LD PLC11_137_step  ; PLC11步137
ANDNOT B_SYS_hold  ; 系统暂停（总）
AND P_On
SET PLC11_138_step  ; PLC11步138
RSET PLC11_137_step  ; PLC11步137

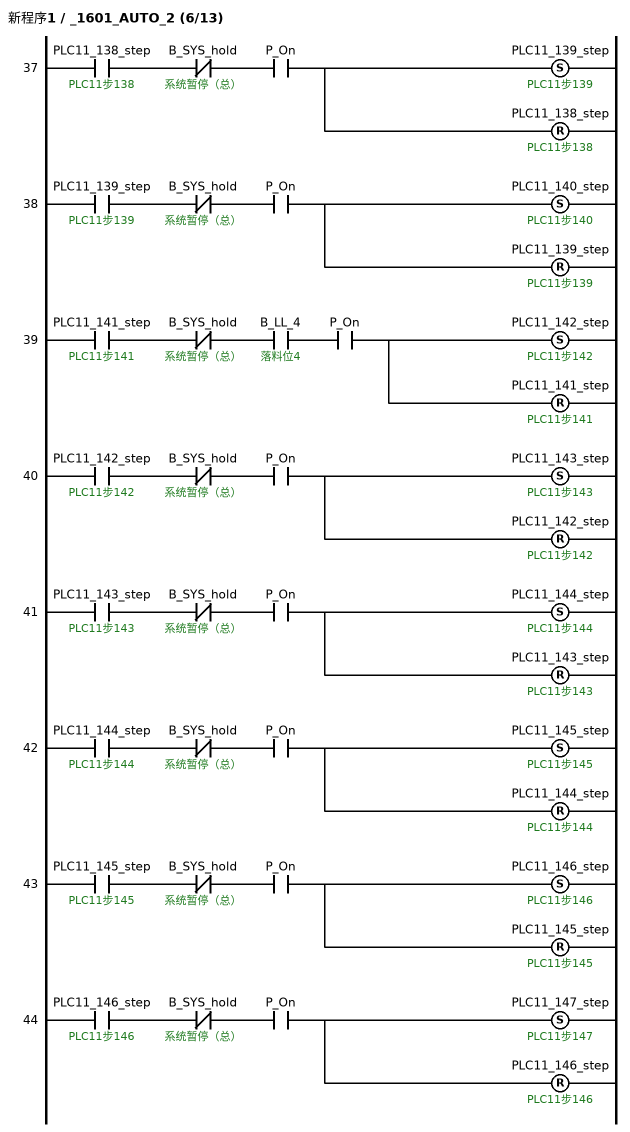
; rung 37
LD PLC11_138_step  ; PLC11步138
ANDNOT B_SYS_hold  ; 系统暂停（总）
AND P_On
SET PLC11_139_step  ; PLC11步139
RSET PLC11_138_step  ; PLC11步138
; rung 38
LD PLC11_139_step  ; PLC11步139
ANDNOT B_SYS_hold  ; 系统暂停（总）
AND P_On
SET PLC11_140_step  ; PLC11步140
RSET PLC11_139_step  ; PLC11步139
; rung 39
LD PLC11_141_step  ; PLC11步141
ANDNOT B_SYS_hold  ; 系统暂停（总）
AND B_LL_4  ; 落料位4
AND P_On
SET PLC11_142_step  ; PLC11步142
RSET PLC11_141_step  ; PLC11步141
; rung 40
LD PLC11_142_step  ; PLC11步142
ANDNOT B_SYS_hold  ; 系统暂停（总）
AND P_On
SET PLC11_143_step  ; PLC11步143
RSET PLC11_142_step  ; PLC11步142
; rung 41
LD PLC11_143_step  ; PLC11步143
ANDNOT B_SYS_hold  ; 系统暂停（总）
AND P_On
SET PLC11_144_step  ; PLC11步144
RSET PLC11_143_step  ; PLC11步143
; rung 42
LD PLC11_144_step  ; PLC11步144
ANDNOT B_SYS_hold  ; 系统暂停（总）
AND P_On
SET PLC11_145_step  ; PLC11步145
RSET PLC11_144_step  ; PLC11步144
; rung 43
LD PLC11_145_step  ; PLC11步145
ANDNOT B_SYS_hold  ; 系统暂停（总）
AND P_On
SET PLC11_146_step  ; PLC11步146
RSET PLC11_145_step  ; PLC11步145
; rung 44
LD PLC11_146_step  ; PLC11步146
ANDNOT B_SYS_hold  ; 系统暂停（总）
AND P_On
SET PLC11_147_step  ; PLC11步147
RSET PLC11_146_step  ; PLC11步146

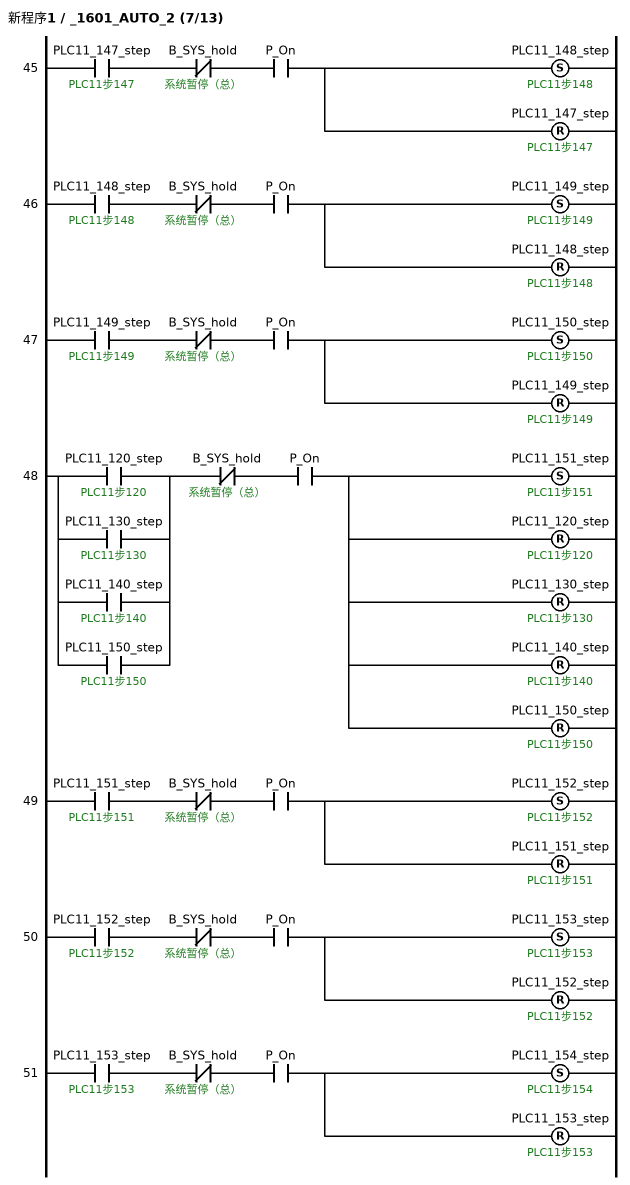
; rung 45
LD PLC11_147_step  ; PLC11步147
ANDNOT B_SYS_hold  ; 系统暂停（总）
AND P_On
SET PLC11_148_step  ; PLC11步148
RSET PLC11_147_step  ; PLC11步147
; rung 46
LD PLC11_148_step  ; PLC11步148
ANDNOT B_SYS_hold  ; 系统暂停（总）
AND P_On
SET PLC11_149_step  ; PLC11步149
RSET PLC11_148_step  ; PLC11步148
; rung 47
LD PLC11_149_step  ; PLC11步149
ANDNOT B_SYS_hold  ; 系统暂停（总）
AND P_On
SET PLC11_150_step  ; PLC11步150
RSET PLC11_149_step  ; PLC11步149
; rung 48
LD PLC11_120_step  ; PLC11步120
OR PLC11_130_step  ; PLC11步130
OR PLC11_140_step  ; PLC11步140
OR PLC11_150_step  ; PLC11步150
ANDNOT B_SYS_hold  ; 系统暂停（总）
AND P_On
SET PLC11_151_step  ; PLC11步151
RSET PLC11_120_step  ; PLC11步120
RSET PLC11_130_step  ; PLC11步130
RSET PLC11_140_step  ; PLC11步140
RSET PLC11_150_step  ; PLC11步150
; rung 49
LD PLC11_151_step  ; PLC11步151
ANDNOT B_SYS_hold  ; 系统暂停（总）
AND P_On
SET PLC11_152_step  ; PLC11步152
RSET PLC11_151_step  ; PLC11步151
; rung 50
LD PLC11_152_step  ; PLC11步152
ANDNOT B_SYS_hold  ; 系统暂停（总）
AND P_On
SET PLC11_153_step  ; PLC11步153
RSET PLC11_152_step  ; PLC11步152
; rung 51
LD PLC11_153_step  ; PLC11步153
ANDNOT B_SYS_hold  ; 系统暂停（总）
AND P_On
SET PLC11_154_step  ; PLC11步154
RSET PLC11_153_step  ; PLC11步153

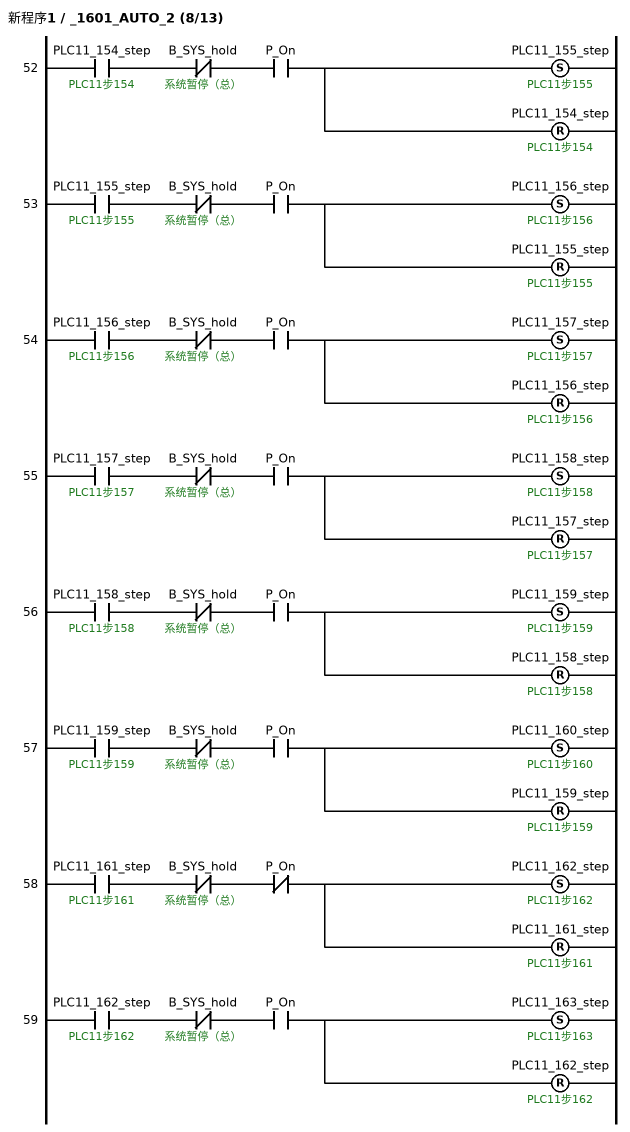
; rung 52
LD PLC11_154_step  ; PLC11步154
ANDNOT B_SYS_hold  ; 系统暂停（总）
AND P_On
SET PLC11_155_step  ; PLC11步155
RSET PLC11_154_step  ; PLC11步154
; rung 53
LD PLC11_155_step  ; PLC11步155
ANDNOT B_SYS_hold  ; 系统暂停（总）
AND P_On
SET PLC11_156_step  ; PLC11步156
RSET PLC11_155_step  ; PLC11步155
; rung 54
LD PLC11_156_step  ; PLC11步156
ANDNOT B_SYS_hold  ; 系统暂停（总）
AND P_On
SET PLC11_157_step  ; PLC11步157
RSET PLC11_156_step  ; PLC11步156
; rung 55
LD PLC11_157_step  ; PLC11步157
ANDNOT B_SYS_hold  ; 系统暂停（总）
AND P_On
SET PLC11_158_step  ; PLC11步158
RSET PLC11_157_step  ; PLC11步157
; rung 56
LD PLC11_158_step  ; PLC11步158
ANDNOT B_SYS_hold  ; 系统暂停（总）
AND P_On
SET PLC11_159_step  ; PLC11步159
RSET PLC11_158_step  ; PLC11步158
; rung 57
LD PLC11_159_step  ; PLC11步159
ANDNOT B_SYS_hold  ; 系统暂停（总）
AND P_On
SET PLC11_160_step  ; PLC11步160
RSET PLC11_159_step  ; PLC11步159
; rung 58
LD PLC11_161_step  ; PLC11步161
ANDNOT B_SYS_hold  ; 系统暂停（总）
ANDNOT P_On
SET PLC11_162_step  ; PLC11步162
RSET PLC11_161_step  ; PLC11步161
; rung 59
LD PLC11_162_step  ; PLC11步162
ANDNOT B_SYS_hold  ; 系统暂停（总）
AND P_On
SET PLC11_163_step  ; PLC11步163
RSET PLC11_162_step  ; PLC11步162

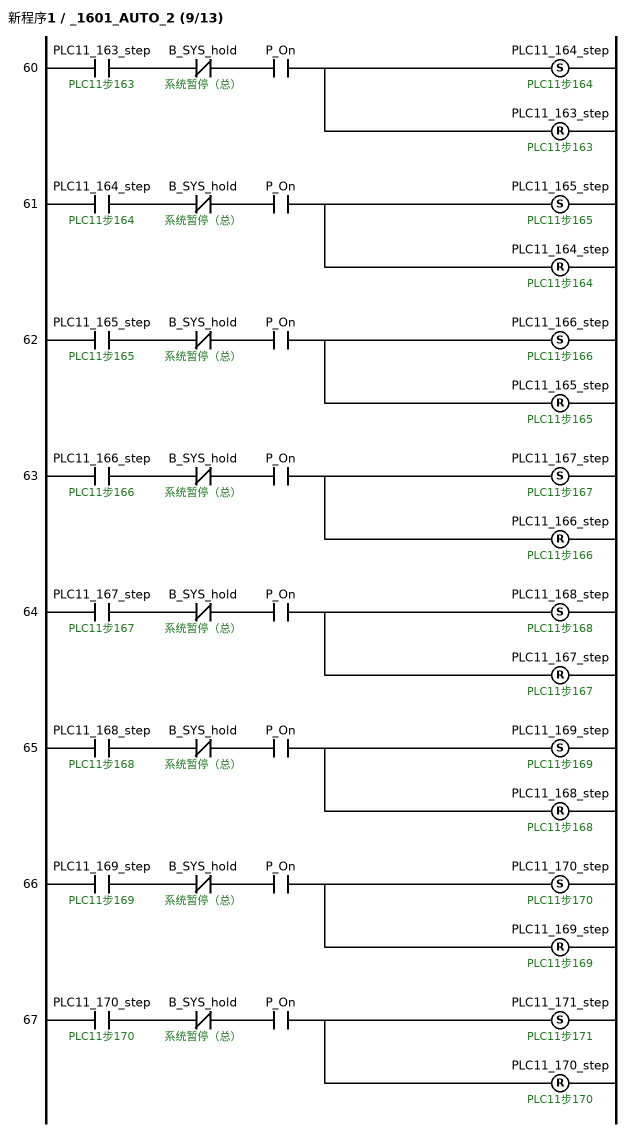
; rung 60
LD PLC11_163_step  ; PLC11步163
ANDNOT B_SYS_hold  ; 系统暂停（总）
AND P_On
SET PLC11_164_step  ; PLC11步164
RSET PLC11_163_step  ; PLC11步163
; rung 61
LD PLC11_164_step  ; PLC11步164
ANDNOT B_SYS_hold  ; 系统暂停（总）
AND P_On
SET PLC11_165_step  ; PLC11步165
RSET PLC11_164_step  ; PLC11步164
; rung 62
LD PLC11_165_step  ; PLC11步165
ANDNOT B_SYS_hold  ; 系统暂停（总）
AND P_On
SET PLC11_166_step  ; PLC11步166
RSET PLC11_165_step  ; PLC11步165
; rung 63
LD PLC11_166_step  ; PLC11步166
ANDNOT B_SYS_hold  ; 系统暂停（总）
AND P_On
SET PLC11_167_step  ; PLC11步167
RSET PLC11_166_step  ; PLC11步166
; rung 64
LD PLC11_167_step  ; PLC11步167
ANDNOT B_SYS_hold  ; 系统暂停（总）
AND P_On
SET PLC11_168_step  ; PLC11步168
RSET PLC11_167_step  ; PLC11步167
; rung 65
LD PLC11_168_step  ; PLC11步168
ANDNOT B_SYS_hold  ; 系统暂停（总）
AND P_On
SET PLC11_169_step  ; PLC11步169
RSET PLC11_168_step  ; PLC11步168
; rung 66
LD PLC11_169_step  ; PLC11步169
ANDNOT B_SYS_hold  ; 系统暂停（总）
AND P_On
SET PLC11_170_step  ; PLC11步170
RSET PLC11_169_step  ; PLC11步169
; rung 67
LD PLC11_170_step  ; PLC11步170
ANDNOT B_SYS_hold  ; 系统暂停（总）
AND P_On
SET PLC11_171_step  ; PLC11步171
RSET PLC11_170_step  ; PLC11步170

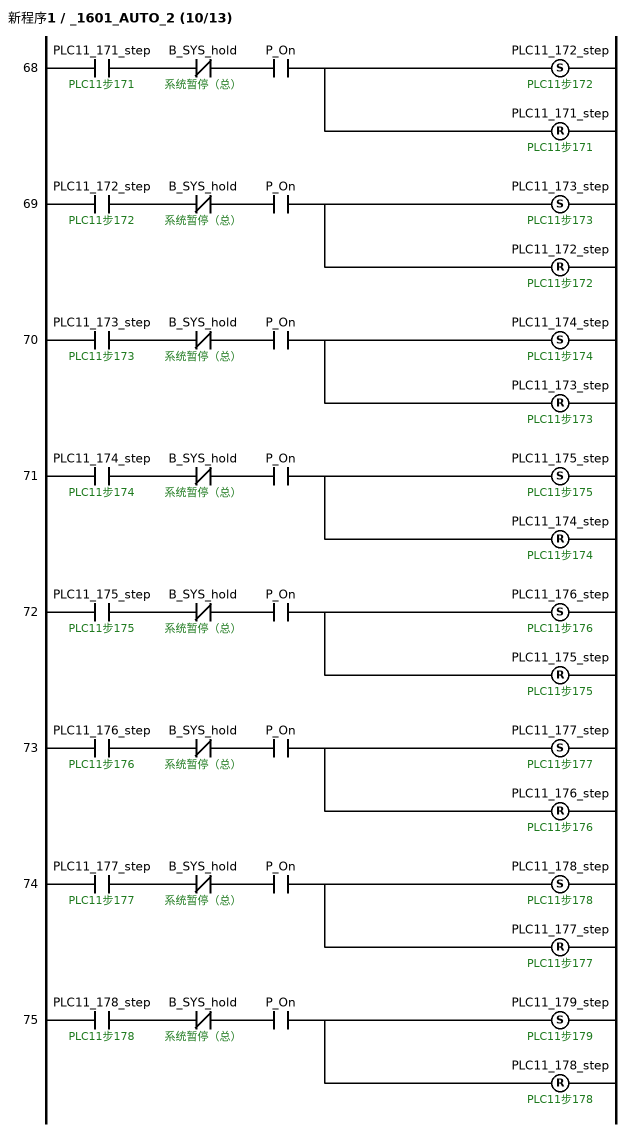
; rung 68
LD PLC11_171_step  ; PLC11步171
ANDNOT B_SYS_hold  ; 系统暂停（总）
AND P_On
SET PLC11_172_step  ; PLC11步172
RSET PLC11_171_step  ; PLC11步171
; rung 69
LD PLC11_172_step  ; PLC11步172
ANDNOT B_SYS_hold  ; 系统暂停（总）
AND P_On
SET PLC11_173_step  ; PLC11步173
RSET PLC11_172_step  ; PLC11步172
; rung 70
LD PLC11_173_step  ; PLC11步173
ANDNOT B_SYS_hold  ; 系统暂停（总）
AND P_On
SET PLC11_174_step  ; PLC11步174
RSET PLC11_173_step  ; PLC11步173
; rung 71
LD PLC11_174_step  ; PLC11步174
ANDNOT B_SYS_hold  ; 系统暂停（总）
AND P_On
SET PLC11_175_step  ; PLC11步175
RSET PLC11_174_step  ; PLC11步174
; rung 72
LD PLC11_175_step  ; PLC11步175
ANDNOT B_SYS_hold  ; 系统暂停（总）
AND P_On
SET PLC11_176_step  ; PLC11步176
RSET PLC11_175_step  ; PLC11步175
; rung 73
LD PLC11_176_step  ; PLC11步176
ANDNOT B_SYS_hold  ; 系统暂停（总）
AND P_On
SET PLC11_177_step  ; PLC11步177
RSET PLC11_176_step  ; PLC11步176
; rung 74
LD PLC11_177_step  ; PLC11步177
ANDNOT B_SYS_hold  ; 系统暂停（总）
AND P_On
SET PLC11_178_step  ; PLC11步178
RSET PLC11_177_step  ; PLC11步177
; rung 75
LD PLC11_178_step  ; PLC11步178
ANDNOT B_SYS_hold  ; 系统暂停（总）
AND P_On
SET PLC11_179_step  ; PLC11步179
RSET PLC11_178_step  ; PLC11步178

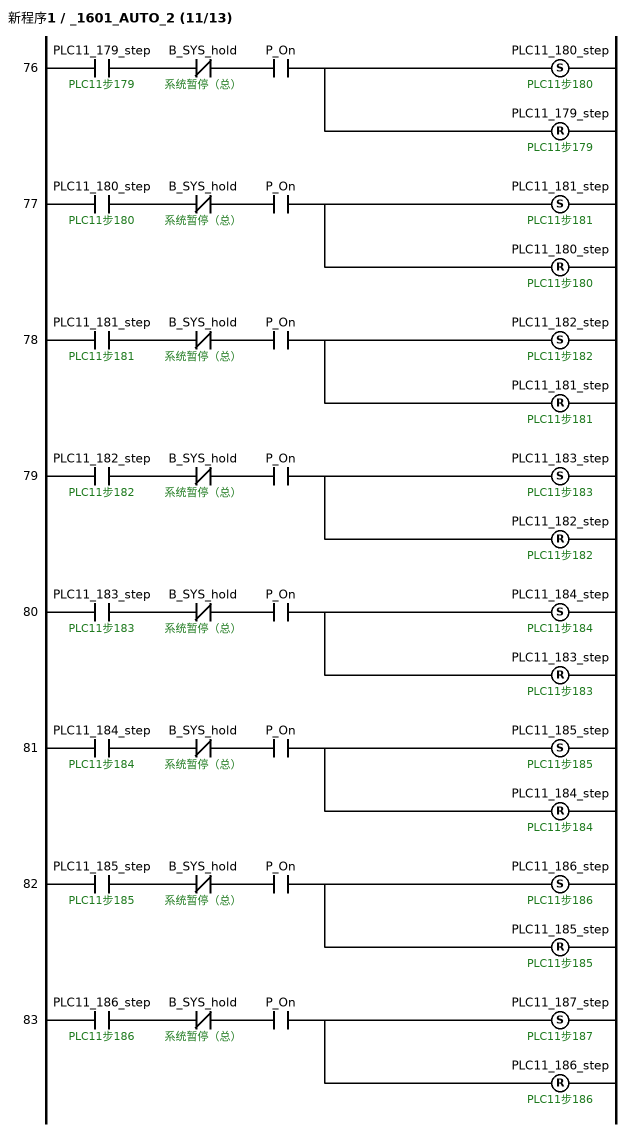
; rung 76
LD PLC11_179_step  ; PLC11步179
ANDNOT B_SYS_hold  ; 系统暂停（总）
AND P_On
SET PLC11_180_step  ; PLC11步180
RSET PLC11_179_step  ; PLC11步179
; rung 77
LD PLC11_180_step  ; PLC11步180
ANDNOT B_SYS_hold  ; 系统暂停（总）
AND P_On
SET PLC11_181_step  ; PLC11步181
RSET PLC11_180_step  ; PLC11步180
; rung 78
LD PLC11_181_step  ; PLC11步181
ANDNOT B_SYS_hold  ; 系统暂停（总）
AND P_On
SET PLC11_182_step  ; PLC11步182
RSET PLC11_181_step  ; PLC11步181
; rung 79
LD PLC11_182_step  ; PLC11步182
ANDNOT B_SYS_hold  ; 系统暂停（总）
AND P_On
SET PLC11_183_step  ; PLC11步183
RSET PLC11_182_step  ; PLC11步182
; rung 80
LD PLC11_183_step  ; PLC11步183
ANDNOT B_SYS_hold  ; 系统暂停（总）
AND P_On
SET PLC11_184_step  ; PLC11步184
RSET PLC11_183_step  ; PLC11步183
; rung 81
LD PLC11_184_step  ; PLC11步184
ANDNOT B_SYS_hold  ; 系统暂停（总）
AND P_On
SET PLC11_185_step  ; PLC11步185
RSET PLC11_184_step  ; PLC11步184
; rung 82
LD PLC11_185_step  ; PLC11步185
ANDNOT B_SYS_hold  ; 系统暂停（总）
AND P_On
SET PLC11_186_step  ; PLC11步186
RSET PLC11_185_step  ; PLC11步185
; rung 83
LD PLC11_186_step  ; PLC11步186
ANDNOT B_SYS_hold  ; 系统暂停（总）
AND P_On
SET PLC11_187_step  ; PLC11步187
RSET PLC11_186_step  ; PLC11步186

